# EPICS substitutions: ioc/PSCApp/Db/out_waveform.substitutions
file db/out_waveform.db {
    pattern {OUT_CHANNEL_NUMBER}
        {"1"}
}
